PROGRAM PRG_06_CrossCut
VAR
	AnalogIn_LREAL_CrossCut: FB_AnalogIn_LREAL;
	lCrossCutMin: LREAL;
	lCrossCutMax: LREAL;
	dCrossCutLeftLimit: DINT;
	dCrossCutRightLimit: DINT;
	
//	dRailLimitLeft: DINT;
//	dRailLimitRight: DINT;

	rCosineAngle: REAL;
	dTeachLimit: DINT;
	rRailHypotenuse: LREAL;
	iRailHypotenuse: DINT;
	dEncoderAddToZero: DINT;
	rTurretOffsetMultiplier: LREAL;
	rCrossCutOffset: REAL;
	rTurretVariable: LREAL;
	rCutSpeed: REAL;
	rReturnSpeed: REAL;
	rDriveMaxSpeed: REAL;
	rBufferSpeed: REAL;
	rSawOFFSpeed: REAL;
	rSpeedScaled: REAL;
	iCrossCutMedianStep: INT;
	R_TRIG_0: R_TRIG;
	R_TRIG_1: R_TRIG;
	RS_CentreTrigger: RS;
	bCentreTrigger: BOOL;
END_VAR

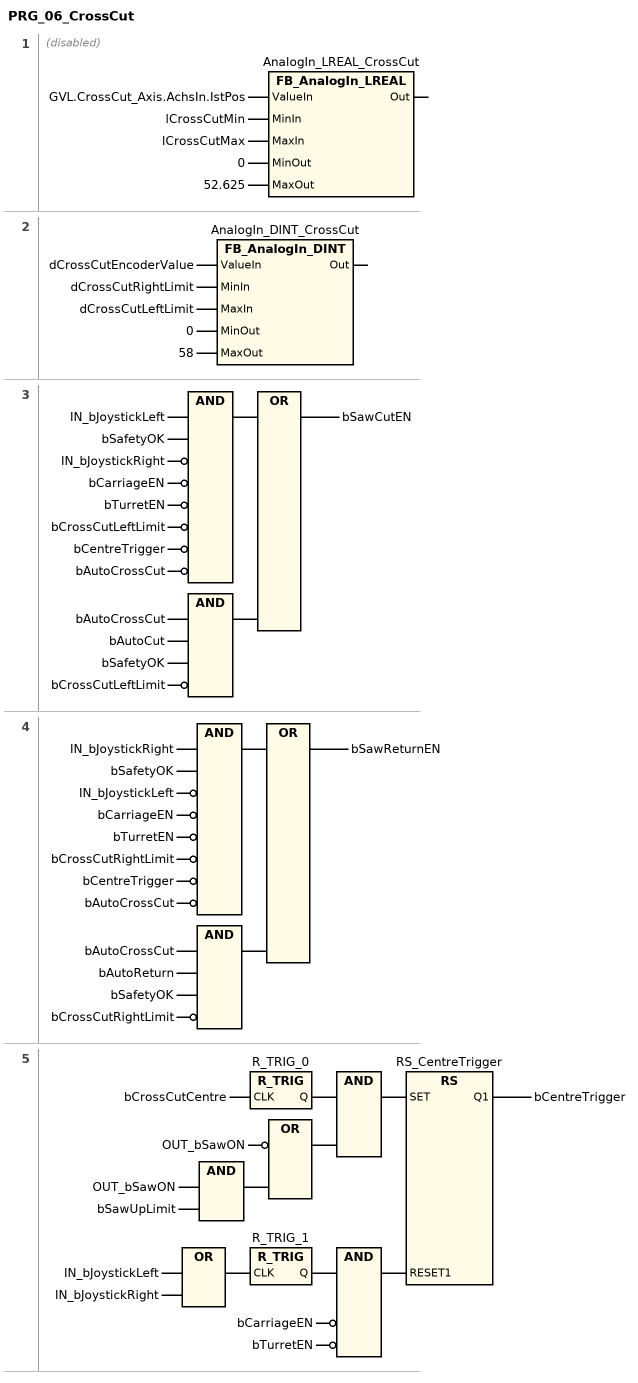
// NETWORK 1 (disabled)
// AnalogIn_LREAL_CrossCut(
//     ValueIn := GVL.CrossCut_Axis.AchsIn.IstPos,
//     MinIn := lCrossCutMin,
//     MaxIn := lCrossCutMax,
//     MinOut := 0,
//     MaxOut := 52.625); // FB_AnalogIn_LREAL

// NETWORK 2
AnalogIn_DINT_CrossCut(
    ValueIn := dCrossCutEncoderValue,
    MinIn := dCrossCutRightLimit,
    MaxIn := dCrossCutLeftLimit,
    MinOut := 0,
    MaxOut := 58); // FB_AnalogIn_DINT

// NETWORK 3
bSawCutEN := IN_bJoystickLeft AND bSafetyOK AND NOT IN_bJoystickRight AND NOT bCarriageEN AND NOT bTurretEN AND NOT bCrossCutLeftLimit AND NOT bCentreTrigger AND NOT bAutoCrossCut OR bAutoCrossCut AND bAutoCut AND bSafetyOK AND NOT bCrossCutLeftLimit;

// NETWORK 4
bSawReturnEN := IN_bJoystickRight AND bSafetyOK AND NOT IN_bJoystickLeft AND NOT bCarriageEN AND NOT bTurretEN AND NOT bCrossCutRightLimit AND NOT bCentreTrigger AND NOT bAutoCrossCut OR bAutoCrossCut AND bAutoReturn AND bSafetyOK AND NOT bCrossCutRightLimit;

// NETWORK 5
R_TRIG_0(CLK := bCrossCutCentre); // R_TRIG
R_TRIG_1(CLK := IN_bJoystickLeft OR IN_bJoystickRight); // R_TRIG
RS_CentreTrigger(SET := R_TRIG_0.Q AND (NOT OUT_bSawON OR OUT_bSawON AND bSawUpLimit), RESET1 := R_TRIG_1.Q AND NOT bCarriageEN AND NOT bTurretEN); // RS
bCentreTrigger := RS_CentreTrigger.Q1;

ACTION ACT_06_1_CrossCut:
//lCrossCutMin := 7050.4087086806794;
//lCrossCutMax := 8385.9641369556011;
dCrossCutLeftLimit := -1251057172 + dEncoderAddToZero;		// move the saw block all the way to the left
dCrossCutRightLimit := -2056805324 + dEncoderAddToZero;  	// move the saw block all the way to the right
dRailLimitLeft := -1321435390 + dEncoderAddToZero;			// align centre of the blade with the left inner edge of the bed rails 
dRailLimitRight := -1986427106 + dEncoderAddToZero;			// align centre of the blade with the right inner edge of the bed rails
dEncoderAddToZero := 2100000000;							// Take the absolute value of the lowest negative number and round up

// Teach Limits left and right
IF bTeachReadyLeft AND bTeach AND bCarriageCentreRef AND bTurretMedianRange AND (AnalogIn_DINT_CrossCut.Out.rScaled > (AnalogIn_DINT_CrossCut.MaxOut / 2)) (*AND NOT (bTurretReturn AND bAutoCrossCut AND bMachineHoming)*) THEN
	dTeachLimitLeft := GVL.PDO_CrossCutAX_IN.A545_AktPosition + dEncoderAddToZero;
ELSIF bTeachReadyRight AND bTeach AND bCarriageCentreRef AND bTurretMedianRange AND (AnalogIn_DINT_CrossCut.Out.rScaled < (AnalogIn_DINT_CrossCut.MaxOut / 2)) (*AND NOT (bTurretReturn AND bAutoCrossCut AND bMachineHoming)*) THEN
	dTeachLimitRight := GVL.PDO_CrossCutAX_IN.A545_AktPosition + dEncoderAddToZero;
END_IF

// CrossCut Limits
IF (dCrossCutEncoderValue >= (dCrossCutMedian + (iRailHypotenuse - dTeachLimit))) OR
	(((AnalogIn_DINT_Turret.Out.rScaled > 85 (*Degrees*)) OR (AnalogIn_DINT_Turret.Out.rScaled < -85)) AND (AnalogIn_DINT_CrossCut.Out.rScaled >= (AnalogIn_DINT_CrossCut.MaxOut - 6 (*Inches*)))) OR
	(dCrossCutEncoderValue > (dCrossCutLeftLimit - 5000))
	THEN
	bCrossCutLeftLimit := TRUE ;	// Left Limit
	bCrossCutRightLimit := FALSE ;
ELSIF (dCrossCutEncoderValue <= (dCrossCutMedian - (iRailHypotenuse - dTeachLimit))) OR
	(((AnalogIn_DINT_Turret.Out.rScaled > 85 (*Degrees*)) OR (AnalogIn_DINT_Turret.Out.rScaled < -85)) AND (AnalogIn_DINT_CrossCut.Out.rScaled <= (AnalogIn_DINT_CrossCut.MinOut + 6 (*Inches*)))) OR
	(dCrossCutEncoderValue < (dCrossCutRightLimit + 5000))
	THEN
	bCrossCutLeftLimit := FALSE ;	
	bCrossCutRightLimit := TRUE ;	// Right Limit
ELSE
	bCrossCutLeftLimit := FALSE ;	
	bCrossCutRightLimit := FALSE ;	
END_IF

// Slowdowns approaching the limits 
IF (dCrossCutEncoderValue >= (dCrossCutMedian + (iRailHypotenuse - dTeachLimit))-50000000) OR
	(((AnalogIn_DINT_Turret.Out.rScaled > 85 (*Degrees*)) OR (AnalogIn_DINT_Turret.Out.rScaled < -85)) AND (AnalogIn_DINT_CrossCut.Out.rScaled >= (AnalogIn_DINT_CrossCut.MaxOut - 6(*Inches*))-1)) OR
	(dCrossCutEncoderValue > (dCrossCutLeftLimit - 50000000))
	THEN
	bApproachingLimitLeft := TRUE ;		// Left approaching limit
	bApproachingLimitRight := FALSE ;
ELSIF (dCrossCutEncoderValue <= (dCrossCutMedian - (iRailHypotenuse - dTeachLimit))+50000000) OR
	(((AnalogIn_DINT_Turret.Out.rScaled > 85 (*Degrees*)) OR (AnalogIn_DINT_Turret.Out.rScaled < -85)) AND (AnalogIn_DINT_CrossCut.Out.rScaled <= (AnalogIn_DINT_CrossCut.MinOut + 6 (*Inches*))+1)) OR
	(dCrossCutEncoderValue < (dCrossCutRightLimit + 50000000))
	THEN
	bApproachingLimitRight := TRUE ;	// Right approaching limit
	bApproachingLimitLeft := FALSE ;	
ELSE
	bApproachingLimitRight := FALSE ;
	bApproachingLimitLeft 	:= FALSE ;
END_IF

// CrossCut encoder rollover code. See Turret's
IF dCrossCutEncoderValue > dCrossCutLeftLimit THEN
	dCrossCutEncoderValue := dCrossCutLeftLimit ;
ELSIF dCrossCutEncoderValue < dCrossCutRightLimit THEN
	dCrossCutEncoderValue := dCrossCutRightLimit ;
ELSE
	dCrossCutEncoderValue := GVL.PDO_CrossCutAX_IN.A545_AktPosition + dEncoderAddToZero ;	
END_IF

// Hypotenuse calculation
IF ABS(AnalogIn_DINT_Turret.Out.rScaled) <> 90 THEN
	rCosineAngle := COS ( (PI / 180) * ABS( AnalogIn_DINT_Turret.Out.rScaled)) ;
ELSE
	rCosineAngle := COS ( (PI / 180) * 89.9999 ) ;
END_IF

dTeachLimit := REAL_TO_DINT(((DINT_TO_REAL(dRailLimitLeft - dRailLimitRight))/2) - ((DINT_TO_REAL(dTeachLimitLeft - dTeachLimitRight))/2)) ;

	rRailHypotenuse := ( (DINT_TO_LREAL(dRailLimitLeft - dRailLimitRight)/2) / rCosineAngle);

IF rRailHypotenuse >= 1942843775 OR rRailHypotenuse < 0 THEN
	iRailHypotenuse := 1942843775;		// rRailHypotenuse = 1942843775 	@ 80°
ELSE
	iRailHypotenuse := LREAL_TO_DINT(rRailHypotenuse);
END_IF 


(* Crosscut offset relative to Carriage position *)
IF bCarriageCentreRef THEN
	rCrossCutOffset := 0 ;
ELSE
	rCrossCutOffset := ABS(AnalogIn_LREAL_Carriage.Out.rScaled - ((AnalogIn_LREAL_Carriage.MaxOut-AnalogIn_LREAL_Carriage.MinOut)/2))(* + rAddend*) ;
END_IF
	
(* Crosscut median *)
rTurretOffsetMultiplier := (rTurretVariable * (ABS(AnalogIn_DINT_Turret.Out.rScaled)/90)) ;
iCrossCutMedianStep;

IF (bCarriageCentreRef AND NOT bTurretMedianRange AND AnalogIn_DINT_Turret.Out.rScaled >0) OR (NOT bCarriageCentreRef AND (AnalogIn_DINT_Turret.Out.rScaled > 85 OR AnalogIn_DINT_Turret.Out.rScaled < -85)) THEN	
	dCrossCutMedian := REAL_TO_DINT (((DINT_TO_REAL(dTeachLimitLeft + dTeachLimitRight)) / 2 ) -  ((rTurretOffsetMultiplier/(AnalogIn_DINT_CrossCut.MaxOut-AnalogIn_DINT_CrossCut.MinOut))*DINT_TO_REAL(dCrossCutLeftLimit-dCrossCutRightLimit))  ) ;
	rTurretVariable := 0.5;
	iCrossCutMedianStep := 10;
ELSIF (bCarriageCentreRef AND NOT bTurretMedianRange AND AnalogIn_DINT_Turret.Out.rScaled <0) OR (NOT bCarriageCentreRef AND (AnalogIn_DINT_Turret.Out.rScaled > 85 OR AnalogIn_DINT_Turret.Out.rScaled < -85)) THEN	
	dCrossCutMedian := REAL_TO_DINT (((DINT_TO_REAL(dTeachLimitLeft + dTeachLimitRight)) / 2 ) +  ((rTurretOffsetMultiplier/(AnalogIn_DINT_CrossCut.MaxOut-AnalogIn_DINT_CrossCut.MinOut))*DINT_TO_REAL(dCrossCutLeftLimit-dCrossCutRightLimit))  ) ;
	rTurretVariable := 0.5;
	iCrossCutMedianStep := 20;
ELSIF NOT bCarriageCentreRef AND (AnalogIn_LREAL_Carriage.Out.rScaled < rCarriageMedian) AND NOT (AnalogIn_DINT_Turret.Out.rScaled > 85 OR AnalogIn_DINT_Turret.Out.rScaled < -85) THEN
	dCrossCutMedian := REAL_TO_DINT(((DINT_TO_REAL(dTeachLimitLeft + dTeachLimitRight)) / 2 ) - ((rCrossCutOffset/(AnalogIn_DINT_CrossCut.MaxOut-AnalogIn_DINT_CrossCut.MinOut))*DINT_TO_REAL(dCrossCutLeftLimit-dCrossCutRightLimit)) /rCosineAngle) ;
	iCrossCutMedianStep := 30;
ELSIF NOT bCarriageCentreRef AND (AnalogIn_LREAL_Carriage.Out.rScaled > rCarriageMedian) AND NOT (AnalogIn_DINT_Turret.Out.rScaled > 85 OR AnalogIn_DINT_Turret.Out.rScaled < -85) THEN
	dCrossCutMedian := REAL_TO_DINT(((DINT_TO_REAL(dTeachLimitLeft + dTeachLimitRight)) / 2 ) + ((rCrossCutOffset/(AnalogIn_DINT_CrossCut.MaxOut-AnalogIn_DINT_CrossCut.MinOut))*DINT_TO_REAL(dCrossCutLeftLimit-dCrossCutRightLimit)) /rCosineAngle) ;
	iCrossCutMedianStep := 40;
END_IF

IF (dCrossCutEncoderValue >= (dCrossCutMedian - 3000000)) AND (dCrossCutEncoderValue <= (dCrossCutMedian + 3000000)) THEN
	bCrossCutCentre := TRUE ;
ELSE
	bCrossCutCentre := FALSE ;
END_IF
END_ACTION

ACTION ACT_06_2_CrossCutSpeed:
rCutSpeed := 20 ;
rReturnSpeed := 75 ;		
rDriveMaxSpeed := 75 ;
rBufferSpeed := 10 ;
rSawOFFSpeed := 75 ;

// Crosscut speed relative to saw blade current feedback
rCrossCutSpeedMultiplier := 1 ;

// Cut and Return speed
IF bSawReturnEN AND NOT bSawCutEN AND NOT bApproachingLimitRight AND OUT_bSawON THEN	// Return speed if Saw blade is ON
	rCrossCutJogVelocity := rReturnSpeed  ;
																	
ELSIF bSawCutEN AND NOT bSawReturnEN AND NOT bApproachingLimitLeft AND OUT_bSawON THEN	// Cut speed if Saw blade is ON
	rCrossCutJogVelocity := (rCutSpeed * rCrossCutSpeedMultiplier) ; // ##### CURRENT FEEDBACK #####
	
ELSIF ((bSawCutEN AND bApproachingLimitLeft) OR (bSawReturnEN AND bApproachingLimitRight))  THEN	// Buffer speed as the blade approaches the edge limits
	rCrossCutJogVelocity := rBufferSpeed ;
	
ELSIF ((bSawCutEN AND NOT bApproachingLimitLeft) OR (bSawReturnEN AND NOT bApproachingLimitRight)) AND NOT OUT_bSawON THEN // Cut and Return speed if Saw blade OFF
	rCrossCutJogVelocity := rSawOFFSpeed ;
(*ELSE
	rCrossCutJogVelocity := 0 ;*)
END_IF
END_ACTION

END_PROGRAM

(* stored: Version 1.1.0.1, ProductVersion 3.1.4024.15
   POU PRG_06_CrossCut: Id {1ada790c-430f-40ff-84a5-63abddfc2ca8}, SpecialFunc None
   Action ACT_06_1_CrossCut: Id {b853cd1c-1170-41a5-a74a-8e2fb720ba0b}
   Action ACT_06_2_CrossCutSpeed: Id {4034cf41-a875-45a4-9ad9-3cc174c2aa10} *)
